PROGRAM PRG_Log_Main

VAR
	logger : FB_SysLogLIstener;
END_VAR

logger.CyclicLogic();

END_PROGRAM

(* stored: Version 1.1.0.1
   POU PRG_Log_Main: Id {bb1d0e3f-e339-4d05-b071-4015d4af0ed5}, SpecialFunc None *)
